TYPE RGI_14_CMD :
(
	Nodef,
	///夹紧指令
	Cmd_Clamp,
	///松开指令
	Cmd_Release,
	///绝对旋转夹紧指令
	Cmd_RotateAbsClamp,
	///绝对旋转松开指令
	Cmd_RotateAbsRelease,
	///增量旋转夹紧指令
	Cmd_RoratRelClamp,
	///增量旋转松开指令
	Cmd_RoratRelRelease,
	///Cmd_Stop,//停止指令
	///初始化指令
	Cmd_Org
);
END_TYPE

(* stored: Version 1.1.0.1, ProductVersion 3.1.4024.9
   DUT RGI_14_CMD: Id {a81d7c8a-734a-47eb-9fbd-98e37ec073c8} *)
